FUNCTION_BLOCK BaseCarrier EXTENDS BaseComponent
VAR_INPUT
END_VAR
VAR_OUTPUT
END_VAR
VAR
	Motor : Motor;
END_VAR

END_FUNCTION_BLOCK

(* stored: Version 1.1.0.1
   POU BaseCarrier: Id {e9ecffdb-cd9d-4d21-8229-51ae00899c07}, SpecialFunc None *)
